// TIA Portal V19 export
TYPE "PosFbk_RTN"
// stored: Access Published
   STRUCT
      Preset : Struct
         Pulses : DInt;
         Units : LReal;
      END_STRUCT;
      Config : Struct
         Resolution : LReal;   // mm/turn or mm/pulse
      END_STRUCT;
   END_STRUCT;
END_TYPE
